PROGRAM IntakeBuffer
VAR
	bInterlocksOK			:BOOL;
	rRealPosition			:REAL;
	rNextPosition			:REAL;
END_VAR
VAR_OUTPUT
	iStep					:UINT;
	iStepTemp				:UINT;
	iPosition				:UINT;
END_VAR

CASE iPosition OF
	0:

		rNextPosition := 2;
	1:
	
		rNextPosition := 3;
	2:

		rNextPosition := 4;
	3:

		rNextPosition := 5;
	4:

		rNextPosition := 6;
	5:

		rNextPosition := 7;
	6:
	
		rNextPosition := 8;
	7:
		rNextPosition := 9;
	8:
		
		rNextPosition := 10;
	9:
		
		rNextPosition := 11;
	10:
		
		rNextPosition := 1;
		
END_CASE

bInterlocksOK := TRUE;

iStepTemp:=iStep;
CASE iStep OF
	0: //Hold
		IF Station.stControl.bRunning THEN
			iStep := 100;
		END_IF
		
	100: //Counting trays
		IF iPosition <= 10 AND IN.bSensor_TrayInReady THEN
			iStep := 400; //Continue
		ELSIF iPosition = 10 AND NOT IN.bSensor_TrayInReady THEN
			iStep := 200; //Buffer empty
		END_IF
	
	200: //Home buffer
		IF IN.bIntakeBuffer_Homed THEN
			iStep := 300;
		END_IF
	
	300: //Call operator and pause process (in MachineControl)
		//Call operator
		iStep := 999;
	
		
	400: //Waiting for Robot
		
		
	500: //Waiting for conveyor
		IF Conveyor.iStep = 999 THEN
			iStep := 600;
		END_IF
		
	600: //Lowering
		IF rRealPosition = rNextPosition THEN 
			iPosition := iPosition + 1;
			iStep := 999;
		END_IF
	
	999: //finish
		iStep := 0;

END_CASE
IF NOT bInterlocksOK THEN
	iStep:=iStepTemp;
END_IF

//Control
//Station.stAutoCmd.bIntakeLift_HOME := F_StepCMP(iStep, 200, 0, 0, 0, 0, 0, 0, 0, 0, 0);
//Station.stAutoCmd.bIntakeLift_DOWN := F_StepCMP(iStep, 600, 0, 0, 0, 0, 0, 0, 0, 0, 0);

END_PROGRAM

(* stored: Version 1.1.0.1
   POU IntakeBuffer: Id {5ff5bb1c-2e49-4a66-b9b8-88b19cd5edbe}, SpecialFunc None *)
